// TIA Portal V21 export
DATA_BLOCK "TimerZona"   // DB45
{ S7_Optimized_Access := 'TRUE' }
// stored: MemoryReserve 100
   VAR RETAIN
      DeltaP_Filtri : "Std_stTimer";
   END_VAR
   VAR
      DeltaT_UscitaSterilizzazione { S7_SetPoint := 'True'} : "Std_stTimer";
      DeltaT_UscitaSosta { S7_SetPoint := 'True'} : "Std_stTimer";
   END_VAR
BEGIN
   DeltaP_Filtri.IN := FALSE;
   DeltaP_Filtri.O := FALSE;
   DeltaP_Filtri.Preset := 5.0;
   DeltaP_Filtri.TempoTrascorso := 0.0;
   DeltaT_UscitaSterilizzazione.IN := FALSE;
   DeltaT_UscitaSterilizzazione.O := FALSE;
   DeltaT_UscitaSterilizzazione.Preset := 5.0;
   DeltaT_UscitaSterilizzazione.TempoTrascorso := 0.0;
   DeltaT_UscitaSosta.IN := FALSE;
   DeltaT_UscitaSosta.O := FALSE;
   DeltaT_UscitaSosta.Preset := 5.0;
   DeltaT_UscitaSosta.TempoTrascorso := 0.0;
END_DATA_BLOCK
